SYSTEM LeGo2_0
  (* Version 1.0, Author, 4DIAC-Consortium *)
  APPLICATION HMI
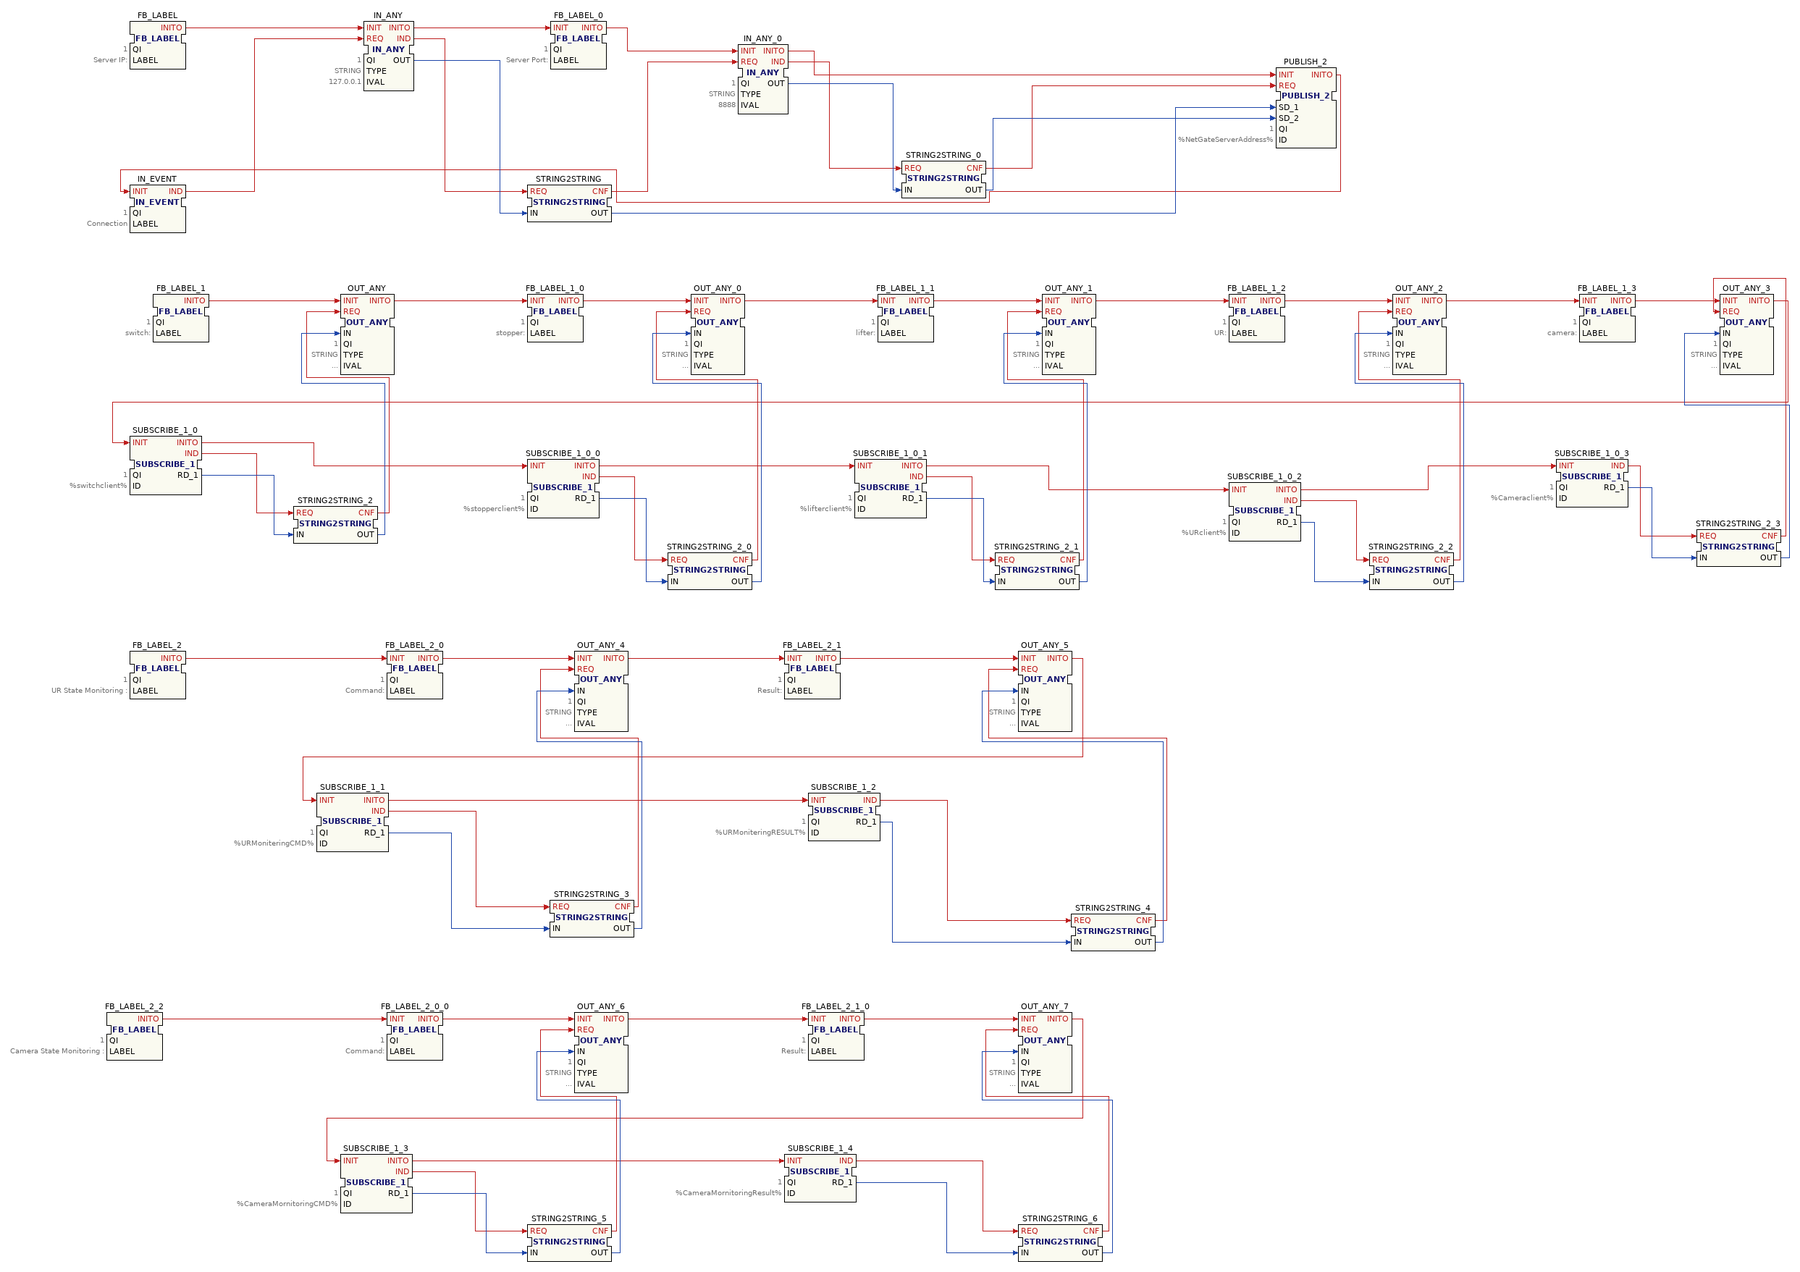
    FBS
      FB_LABEL : FB_LABEL(QI := 1, LABEL := Server IP:);
      FB_LABEL_0 : FB_LABEL(QI := 1, LABEL := Server Port:);
      IN_ANY : IN_ANY(QI := 1, TYPE := STRING, IVAL := 127.0.0.1);
      IN_ANY_0 : IN_ANY(QI := 1, TYPE := STRING, IVAL := 8888);
      PUBLISH_2 : PUBLISH_2(QI := 1, ID := %NetGateServerAddress%);
      STRING2STRING : STRING2STRING;
      STRING2STRING_0 : STRING2STRING;
      IN_EVENT : IN_EVENT(QI := 1, LABEL := Connection);
      FB_LABEL_1 : FB_LABEL(QI := 1, LABEL := switch:);
      FB_LABEL_1_0 : FB_LABEL(QI := 1, LABEL := stopper:);
      FB_LABEL_1_1 : FB_LABEL(QI := 1, LABEL := lifter:);
      FB_LABEL_1_2 : FB_LABEL(QI := 1, LABEL := UR:);
      FB_LABEL_1_3 : FB_LABEL(QI := 1, LABEL := camera:);
      OUT_ANY : OUT_ANY(QI := 1, TYPE := STRING, IVAL := ...);
      OUT_ANY_0 : OUT_ANY(QI := 1, TYPE := STRING, IVAL := ...);
      OUT_ANY_1 : OUT_ANY(QI := 1, TYPE := STRING, IVAL := ...);
      OUT_ANY_2 : OUT_ANY(QI := 1, TYPE := STRING, IVAL := ...);
      OUT_ANY_3 : OUT_ANY(QI := 1, TYPE := STRING, IVAL := ...);
      SUBSCRIBE_1_0 : SUBSCRIBE_1(QI := 1, ID := %switchclient%);
      SUBSCRIBE_1_0_0 : SUBSCRIBE_1(QI := 1, ID := %stopperclient%);
      SUBSCRIBE_1_0_1 : SUBSCRIBE_1(QI := 1, ID := %lifterclient%);
      SUBSCRIBE_1_0_2 : SUBSCRIBE_1(QI := 1, ID := %URclient%);
      SUBSCRIBE_1_0_3 : SUBSCRIBE_1(QI := 1, ID := %Cameraclient%);
      STRING2STRING_2 : STRING2STRING;
      STRING2STRING_2_0 : STRING2STRING;
      STRING2STRING_2_1 : STRING2STRING;
      STRING2STRING_2_2 : STRING2STRING;
      STRING2STRING_2_3 : STRING2STRING;
      FB_LABEL_2 : FB_LABEL(QI := 1, LABEL := UR State Monitoring :);
      FB_LABEL_2_0 : FB_LABEL(QI := 1, LABEL := Command:);
      FB_LABEL_2_1 : FB_LABEL(QI := 1, LABEL := Result:);
      FB_LABEL_2_2 : FB_LABEL(QI := 1, LABEL := Camera State Monitoring :);
      FB_LABEL_2_0_0 : FB_LABEL(QI := 1, LABEL := Command:);
      FB_LABEL_2_1_0 : FB_LABEL(QI := 1, LABEL := Result:);
      OUT_ANY_4 : OUT_ANY(QI := 1, TYPE := STRING, IVAL := ...);
      OUT_ANY_5 : OUT_ANY(QI := 1, TYPE := STRING, IVAL := ...);
      OUT_ANY_6 : OUT_ANY(QI := 1, TYPE := STRING, IVAL := ...);
      OUT_ANY_7 : OUT_ANY(QI := 1, TYPE := STRING, IVAL := ...);
      SUBSCRIBE_1_1 : SUBSCRIBE_1(QI := 1, ID := %URMoniteringCMD%);
      SUBSCRIBE_1_2 : SUBSCRIBE_1(QI := 1, ID := %URMoniteringRESULT%);
      SUBSCRIBE_1_3 : SUBSCRIBE_1(QI := 1, ID := %CameraMornitoringCMD%);
      SUBSCRIBE_1_4 : SUBSCRIBE_1(QI := 1, ID := %CameraMornitoringResult%);
      STRING2STRING_3 : STRING2STRING;
      STRING2STRING_4 : STRING2STRING;
      STRING2STRING_5 : STRING2STRING;
      STRING2STRING_6 : STRING2STRING;
    END_FBS
    EVENT_CONNECTIONS
      FB_LABEL.INITO TO IN_ANY.INIT;
      IN_ANY.INITO TO FB_LABEL_0.INIT;
      FB_LABEL_0.INITO TO IN_ANY_0.INIT;
      IN_ANY_0.INITO TO PUBLISH_2.INIT;
      IN_ANY.IND TO STRING2STRING.REQ;
      STRING2STRING.CNF TO IN_ANY_0.REQ;
      IN_ANY_0.IND TO STRING2STRING_0.REQ;
      STRING2STRING_0.CNF TO PUBLISH_2.REQ;
      IN_EVENT.IND TO IN_ANY.REQ;
      PUBLISH_2.INITO TO IN_EVENT.INIT;
      FB_LABEL_1.INITO TO OUT_ANY.INIT;
      OUT_ANY.INITO TO FB_LABEL_1_0.INIT;
      FB_LABEL_1_0.INITO TO OUT_ANY_0.INIT;
      OUT_ANY_0.INITO TO FB_LABEL_1_1.INIT;
      FB_LABEL_1_1.INITO TO OUT_ANY_1.INIT;
      OUT_ANY_1.INITO TO FB_LABEL_1_2.INIT;
      FB_LABEL_1_2.INITO TO OUT_ANY_2.INIT;
      OUT_ANY_2.INITO TO FB_LABEL_1_3.INIT;
      FB_LABEL_1_3.INITO TO OUT_ANY_3.INIT;
      OUT_ANY_3.INITO TO SUBSCRIBE_1_0.INIT;
      SUBSCRIBE_1_0.INITO TO SUBSCRIBE_1_0_0.INIT;
      SUBSCRIBE_1_0_0.INITO TO SUBSCRIBE_1_0_1.INIT;
      SUBSCRIBE_1_0_1.INITO TO SUBSCRIBE_1_0_2.INIT;
      SUBSCRIBE_1_0_2.INITO TO SUBSCRIBE_1_0_3.INIT;
      SUBSCRIBE_1_0.IND TO STRING2STRING_2.REQ;
      STRING2STRING_2.CNF TO OUT_ANY.REQ;
      SUBSCRIBE_1_0_0.IND TO STRING2STRING_2_0.REQ;
      STRING2STRING_2_0.CNF TO OUT_ANY_0.REQ;
      SUBSCRIBE_1_0_1.IND TO STRING2STRING_2_1.REQ;
      STRING2STRING_2_1.CNF TO OUT_ANY_1.REQ;
      SUBSCRIBE_1_0_2.IND TO STRING2STRING_2_2.REQ;
      STRING2STRING_2_2.CNF TO OUT_ANY_2.REQ;
      SUBSCRIBE_1_0_3.IND TO STRING2STRING_2_3.REQ;
      STRING2STRING_2_3.CNF TO OUT_ANY_3.REQ;
      FB_LABEL_2.INITO TO FB_LABEL_2_0.INIT;
      FB_LABEL_2_0.INITO TO OUT_ANY_4.INIT;
      OUT_ANY_4.INITO TO FB_LABEL_2_1.INIT;
      FB_LABEL_2_1.INITO TO OUT_ANY_5.INIT;
      FB_LABEL_2_2.INITO TO FB_LABEL_2_0_0.INIT;
      FB_LABEL_2_0_0.INITO TO OUT_ANY_6.INIT;
      OUT_ANY_6.INITO TO FB_LABEL_2_1_0.INIT;
      FB_LABEL_2_1_0.INITO TO OUT_ANY_7.INIT;
      OUT_ANY_5.INITO TO SUBSCRIBE_1_1.INIT;
      SUBSCRIBE_1_1.INITO TO SUBSCRIBE_1_2.INIT;
      SUBSCRIBE_1_1.IND TO STRING2STRING_3.REQ;
      STRING2STRING_3.CNF TO OUT_ANY_4.REQ;
      SUBSCRIBE_1_2.IND TO STRING2STRING_4.REQ;
      STRING2STRING_4.CNF TO OUT_ANY_5.REQ;
      OUT_ANY_7.INITO TO SUBSCRIBE_1_3.INIT;
      SUBSCRIBE_1_3.INITO TO SUBSCRIBE_1_4.INIT;
      SUBSCRIBE_1_3.IND TO STRING2STRING_5.REQ;
      STRING2STRING_5.CNF TO OUT_ANY_6.REQ;
      SUBSCRIBE_1_4.IND TO STRING2STRING_6.REQ;
      STRING2STRING_6.CNF TO OUT_ANY_7.REQ;
    END_CONNECTIONS
    DATA_CONNECTIONS
      IN_ANY.OUT TO STRING2STRING.IN;
      STRING2STRING.OUT TO PUBLISH_2.SD_1;
      IN_ANY_0.OUT TO STRING2STRING_0.IN;
      STRING2STRING_0.OUT TO PUBLISH_2.SD_2;
      SUBSCRIBE_1_0.RD_1 TO STRING2STRING_2.IN;
      STRING2STRING_2.OUT TO OUT_ANY.IN;
      SUBSCRIBE_1_0_0.RD_1 TO STRING2STRING_2_0.IN;
      STRING2STRING_2_0.OUT TO OUT_ANY_0.IN;
      SUBSCRIBE_1_0_1.RD_1 TO STRING2STRING_2_1.IN;
      STRING2STRING_2_1.OUT TO OUT_ANY_1.IN;
      SUBSCRIBE_1_0_2.RD_1 TO STRING2STRING_2_2.IN;
      STRING2STRING_2_2.OUT TO OUT_ANY_2.IN;
      SUBSCRIBE_1_0_3.RD_1 TO STRING2STRING_2_3.IN;
      STRING2STRING_2_3.OUT TO OUT_ANY_3.IN;
      SUBSCRIBE_1_1.RD_1 TO STRING2STRING_3.IN;
      STRING2STRING_3.OUT TO OUT_ANY_4.IN;
      SUBSCRIBE_1_2.RD_1 TO STRING2STRING_4.IN;
      STRING2STRING_4.OUT TO OUT_ANY_5.IN;
      SUBSCRIBE_1_3.RD_1 TO STRING2STRING_5.IN;
      STRING2STRING_5.OUT TO OUT_ANY_6.IN;
      SUBSCRIBE_1_4.RD_1 TO STRING2STRING_6.IN;
      STRING2STRING_6.OUT TO OUT_ANY_7.IN;
    END_CONNECTIONS
  END_APPLICATION
  APPLICATION SwitchStopperLifter
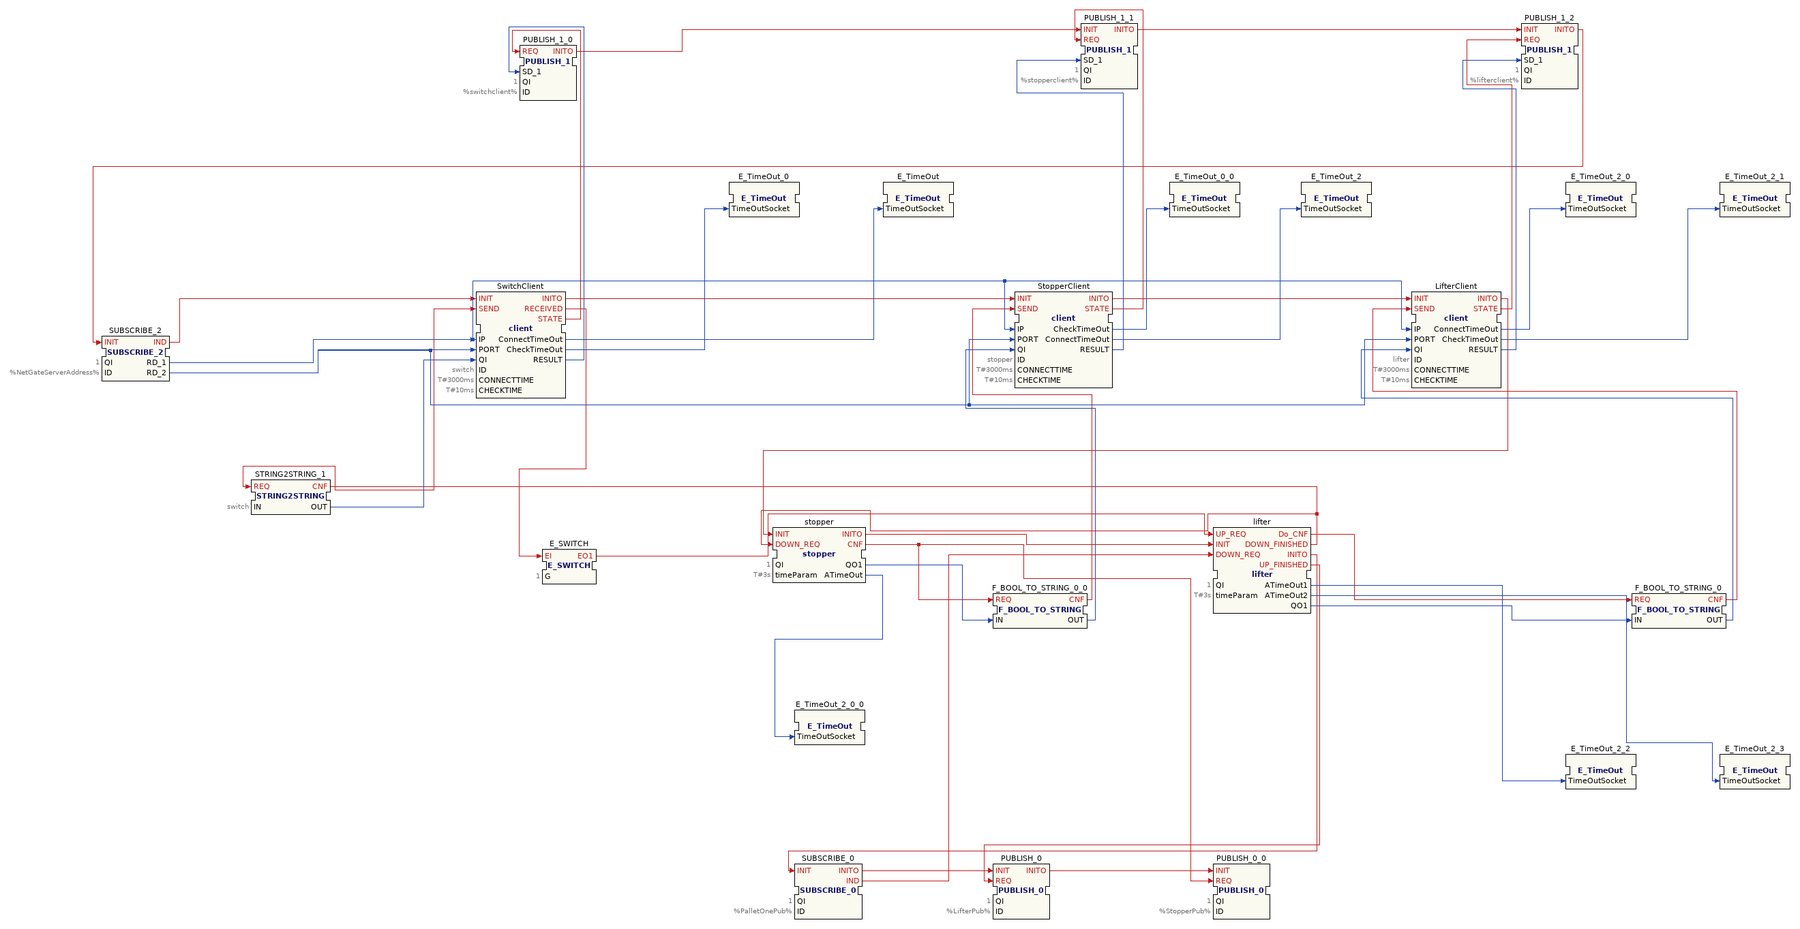
    FBS
      SwitchClient : client(ID := switch, CONNECTTIME := T#3000ms, CHECKTIME := T#10ms);
      E_TimeOut : E_TimeOut;
      E_TimeOut_0 : E_TimeOut;
      SUBSCRIBE_2 : SUBSCRIBE_2(QI := 1, ID := %NetGateServerAddress%);
      LifterClient : client(ID := lifter, CONNECTTIME := T#3000ms, CHECKTIME := T#10ms);
      E_TimeOut_0_0 : E_TimeOut;
      StopperClient : client(ID := stopper, CONNECTTIME := T#3000ms, CHECKTIME := T#10ms);
      E_TimeOut_2 : E_TimeOut;
      E_SWITCH : E_SWITCH(G := 1);
      stopper : stopper(QI := 1, timeParam := T#3s);
      lifter : lifter(QI := 1, timeParam := T#3s);
      E_TimeOut_2_0 : E_TimeOut;
      E_TimeOut_2_1 : E_TimeOut;
      E_TimeOut_2_2 : E_TimeOut;
      E_TimeOut_2_3 : E_TimeOut;
      F_BOOL_TO_STRING_0 : F_BOOL_TO_STRING;
      F_BOOL_TO_STRING_0_0 : F_BOOL_TO_STRING;
      E_TimeOut_2_0_0 : E_TimeOut;
      STRING2STRING_1 : STRING2STRING(IN := switch);
      PUBLISH_0 : PUBLISH_0(QI := 1, ID := %LifterPub%);
      SUBSCRIBE_0 : SUBSCRIBE_0(QI := 1, ID := %PalletOnePub%);
      PUBLISH_0_0 : PUBLISH_0(QI := 1, ID := %StopperPub%);
      PUBLISH_1_0 : PUBLISH_1(QI := 1, ID := %switchclient%);
      PUBLISH_1_1 : PUBLISH_1(QI := 1, ID := %stopperclient%);
      PUBLISH_1_2 : PUBLISH_1(QI := 1, ID := %lifterclient%);
    END_FBS
    EVENT_CONNECTIONS
      SUBSCRIBE_2.IND TO SwitchClient.INIT;
      SwitchClient.INITO TO StopperClient.INIT;
      StopperClient.INITO TO LifterClient.INIT;
      SwitchClient.RECEIVED TO E_SWITCH.EI;
      E_SWITCH.EO1 TO lifter.UP_REQ;
      LifterClient.INITO TO stopper.INIT;
      stopper.INITO TO lifter.INIT;
      lifter.Do_CNF TO F_BOOL_TO_STRING_0.REQ;
      F_BOOL_TO_STRING_0.CNF TO LifterClient.SEND;
      stopper.CNF TO F_BOOL_TO_STRING_0_0.REQ;
      F_BOOL_TO_STRING_0_0.CNF TO StopperClient.SEND;
      lifter.DOWN_FINISHED TO stopper.DOWN_REQ;
      lifter.DOWN_FINISHED TO STRING2STRING_1.REQ;
      STRING2STRING_1.CNF TO SwitchClient.SEND;
      lifter.INITO TO SUBSCRIBE_0.INIT;
      SUBSCRIBE_0.INITO TO PUBLISH_0.INIT;
      SUBSCRIBE_0.IND TO lifter.DOWN_REQ;
      lifter.UP_FINISHED TO PUBLISH_0.REQ;
      PUBLISH_0.INITO TO PUBLISH_0_0.INIT;
      stopper.CNF TO PUBLISH_0_0.REQ;
      PUBLISH_1_0.INITO TO PUBLISH_1_1.INIT;
      PUBLISH_1_1.INITO TO PUBLISH_1_2.INIT;
      PUBLISH_1_2.INITO TO SUBSCRIBE_2.INIT;
      SwitchClient.STATE TO PUBLISH_1_0.REQ;
      StopperClient.STATE TO PUBLISH_1_1.REQ;
      LifterClient.STATE TO PUBLISH_1_2.REQ;
    END_CONNECTIONS
    DATA_CONNECTIONS
      SwitchClient.ConnectTimeOut TO E_TimeOut.TimeOutSocket;
      SwitchClient.CheckTimeOut TO E_TimeOut_0.TimeOutSocket;
      SUBSCRIBE_2.RD_1 TO SwitchClient.IP;
      SUBSCRIBE_2.RD_2 TO SwitchClient.PORT;
      SUBSCRIBE_2.RD_1 TO LifterClient.IP;
      SUBSCRIBE_2.RD_2 TO LifterClient.PORT;
      StopperClient.CheckTimeOut TO E_TimeOut_0_0.TimeOutSocket;
      StopperClient.ConnectTimeOut TO E_TimeOut_2.TimeOutSocket;
      SUBSCRIBE_2.RD_1 TO StopperClient.IP;
      SUBSCRIBE_2.RD_2 TO StopperClient.PORT;
      LifterClient.ConnectTimeOut TO E_TimeOut_2_0.TimeOutSocket;
      LifterClient.CheckTimeOut TO E_TimeOut_2_1.TimeOutSocket;
      lifter.ATimeOut1 TO E_TimeOut_2_2.TimeOutSocket;
      lifter.ATimeOut2 TO E_TimeOut_2_3.TimeOutSocket;
      lifter.QO1 TO F_BOOL_TO_STRING_0.IN;
      F_BOOL_TO_STRING_0.OUT TO LifterClient.QI;
      stopper.QO1 TO F_BOOL_TO_STRING_0_0.IN;
      F_BOOL_TO_STRING_0_0.OUT TO StopperClient.QI;
      stopper.ATimeOut TO E_TimeOut_2_0_0.TimeOutSocket;
      STRING2STRING_1.OUT TO SwitchClient.QI;
      SwitchClient.RESULT TO PUBLISH_1_0.SD_1;
      StopperClient.RESULT TO PUBLISH_1_1.SD_1;
      LifterClient.RESULT TO PUBLISH_1_2.SD_1;
    END_CONNECTIONS
  END_APPLICATION
  APPLICATION URCamera
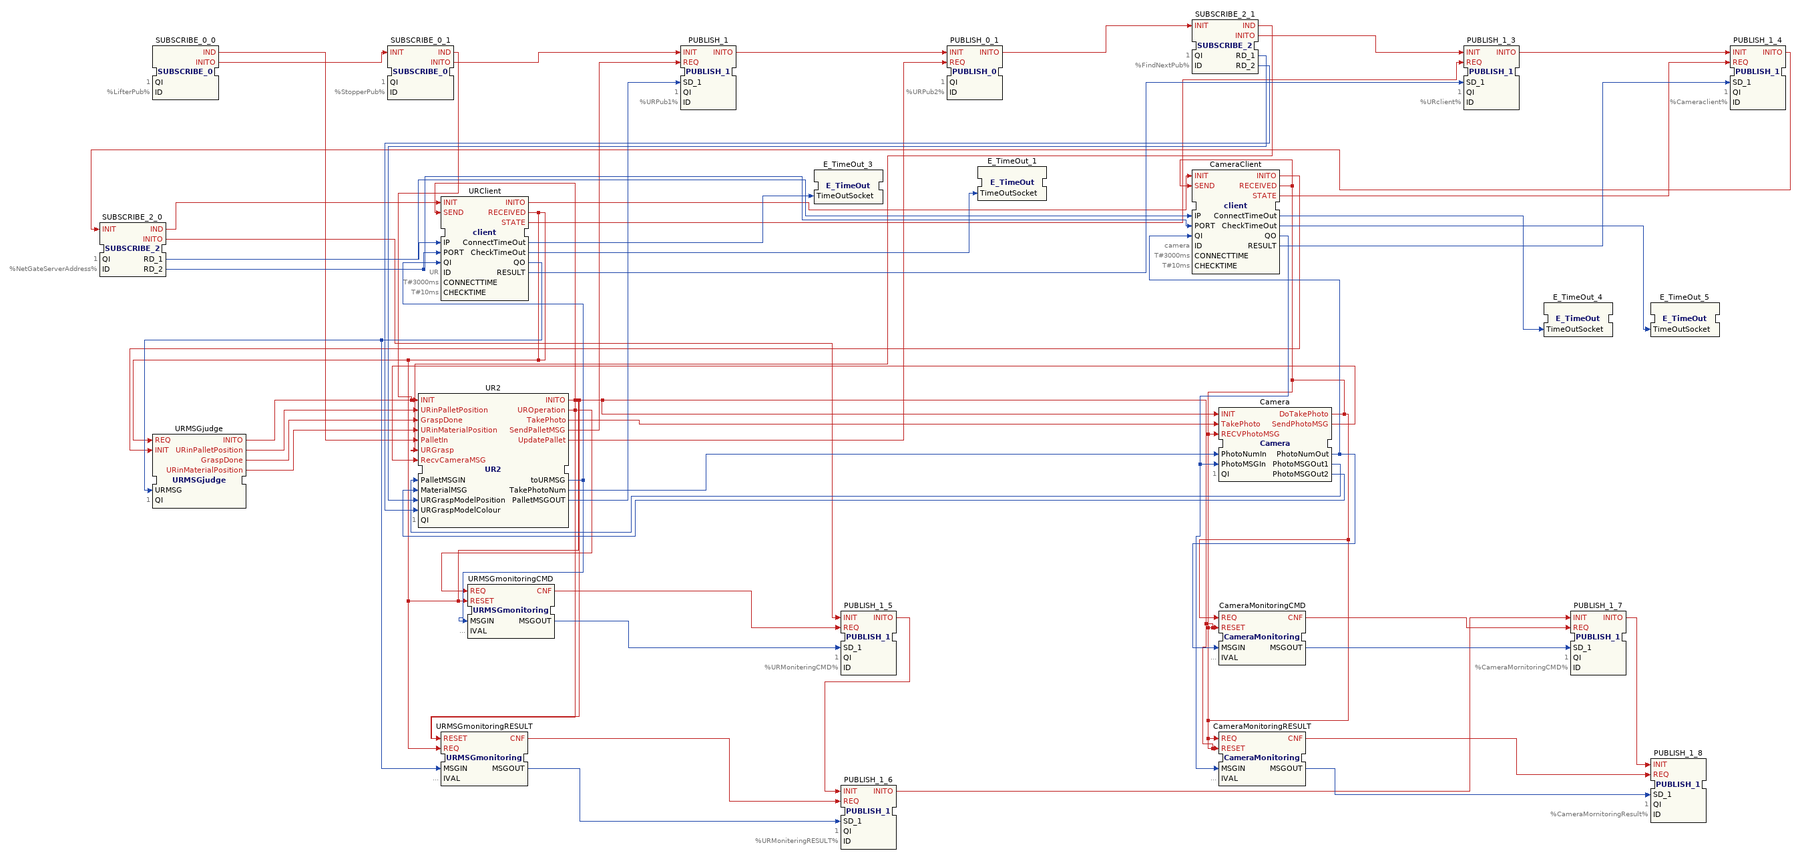
    FBS
      UR2 : UR2(QI := 1);
      URMSGjudge : URMSGjudge(QI := 1);
      URMSGmonitoringRESULT : URMSGmonitoring(IVAL := ...);
      URClient : client(ID := UR, CONNECTTIME := T#3000ms, CHECKTIME := T#10ms);
      E_TimeOut_1 : E_TimeOut;
      E_TimeOut_3 : E_TimeOut;
      Camera : Camera(QI := 1);
      CameraMonitoringCMD : CameraMonitoring(IVAL := ...);
      CameraClient : client(ID := camera, CONNECTTIME := T#3000ms, CHECKTIME := T#10ms);
      E_TimeOut_4 : E_TimeOut;
      E_TimeOut_5 : E_TimeOut;
      SUBSCRIBE_2_0 : SUBSCRIBE_2(QI := 1, ID := %NetGateServerAddress%);
      SUBSCRIBE_0_0 : SUBSCRIBE_0(QI := 1, ID := %LifterPub%);
      SUBSCRIBE_0_1 : SUBSCRIBE_0(QI := 1, ID := %StopperPub%);
      PUBLISH_1 : PUBLISH_1(QI := 1, ID := %URPub1%);
      PUBLISH_0_1 : PUBLISH_0(QI := 1, ID := %URPub2%);
      SUBSCRIBE_2_1 : SUBSCRIBE_2(QI := 1, ID := %FindNextPub%);
      PUBLISH_1_3 : PUBLISH_1(QI := 1, ID := %URclient%);
      PUBLISH_1_4 : PUBLISH_1(QI := 1, ID := %Cameraclient%);
      URMSGmonitoringCMD : URMSGmonitoring(IVAL := ...);
      CameraMonitoringRESULT : CameraMonitoring(IVAL := ...);
      PUBLISH_1_5 : PUBLISH_1(QI := 1, ID := %URMoniteringCMD%);
      PUBLISH_1_6 : PUBLISH_1(QI := 1, ID := %URMoniteringRESULT%);
      PUBLISH_1_7 : PUBLISH_1(QI := 1, ID := %CameraMornitoringCMD%);
      PUBLISH_1_8 : PUBLISH_1(QI := 1, ID := %CameraMornitoringResult%);
    END_FBS
    EVENT_CONNECTIONS
      SUBSCRIBE_2_0.IND TO URClient.INIT;
      URClient.INITO TO CameraClient.INIT;
      URClient.RECEIVED TO URMSGjudge.REQ;
      CameraClient.INITO TO URMSGjudge.INIT;
      URMSGjudge.INITO TO UR2.INIT;
      UR2.INITO TO Camera.INIT;
      URMSGjudge.URinPalletPosition TO UR2.URinPalletPosition;
      URMSGjudge.GraspDone TO UR2.GraspDone;
      URMSGjudge.URinMaterialPosition TO UR2.URinMaterialPosition;
      SUBSCRIBE_0_0.IND TO UR2.PalletIn;
      SUBSCRIBE_0_0.INITO TO SUBSCRIBE_0_1.INIT;
      SUBSCRIBE_0_1.IND TO UR2.INIT;
      UR2.UROperation TO URClient.SEND;
      UR2.TakePhoto TO Camera.TakePhoto;
      Camera.DoTakePhoto TO CameraClient.SEND;
      CameraClient.RECEIVED TO Camera.RECVPhotoMSG;
      SUBSCRIBE_0_1.INITO TO PUBLISH_1.INIT;
      PUBLISH_1.INITO TO PUBLISH_0_1.INIT;
      UR2.SendPalletMSG TO PUBLISH_1.REQ;
      UR2.UpdatePallet TO PUBLISH_0_1.REQ;
      PUBLISH_0_1.INITO TO SUBSCRIBE_2_1.INIT;
      SUBSCRIBE_2_1.IND TO UR2.URGrasp;
      Camera.SendPhotoMSG TO UR2.RecvCameraMSG;
      SUBSCRIBE_2_1.INITO TO PUBLISH_1_3.INIT;
      PUBLISH_1_3.INITO TO PUBLISH_1_4.INIT;
      URClient.STATE TO PUBLISH_1_3.REQ;
      CameraClient.STATE TO PUBLISH_1_4.REQ;
      PUBLISH_1_4.INITO TO SUBSCRIBE_2_0.INIT;
      UR2.UROperation TO URMSGmonitoringCMD.REQ;
      UR2.UROperation TO URMSGmonitoringRESULT.RESET;
      URClient.RECEIVED TO URMSGmonitoringRESULT.REQ;
      URClient.RECEIVED TO URMSGmonitoringCMD.RESET;
      Camera.DoTakePhoto TO CameraMonitoringCMD.REQ;
      CameraClient.RECEIVED TO CameraMonitoringRESULT.REQ;
      Camera.DoTakePhoto TO CameraMonitoringRESULT.RESET;
      CameraClient.RECEIVED TO CameraMonitoringCMD.RESET;
      SUBSCRIBE_2_0.INITO TO PUBLISH_1_5.INIT;
      PUBLISH_1_5.INITO TO PUBLISH_1_6.INIT;
      PUBLISH_1_6.INITO TO PUBLISH_1_7.INIT;
      PUBLISH_1_7.INITO TO PUBLISH_1_8.INIT;
      URMSGmonitoringCMD.CNF TO PUBLISH_1_5.REQ;
      URMSGmonitoringRESULT.CNF TO PUBLISH_1_6.REQ;
      CameraMonitoringCMD.CNF TO PUBLISH_1_7.REQ;
      CameraMonitoringRESULT.CNF TO PUBLISH_1_8.REQ;
      UR2.INITO TO URMSGmonitoringCMD.RESET;
      UR2.INITO TO URMSGmonitoringRESULT.RESET;
      UR2.INITO TO CameraMonitoringCMD.RESET;
      UR2.INITO TO CameraMonitoringRESULT.RESET;
    END_CONNECTIONS
    DATA_CONNECTIONS
      URClient.ConnectTimeOut TO E_TimeOut_3.TimeOutSocket;
      URClient.CheckTimeOut TO E_TimeOut_1.TimeOutSocket;
      CameraClient.ConnectTimeOut TO E_TimeOut_4.TimeOutSocket;
      CameraClient.CheckTimeOut TO E_TimeOut_5.TimeOutSocket;
      SUBSCRIBE_2_0.RD_1 TO URClient.IP;
      SUBSCRIBE_2_0.RD_2 TO URClient.PORT;
      SUBSCRIBE_2_0.RD_1 TO CameraClient.IP;
      SUBSCRIBE_2_0.RD_2 TO CameraClient.PORT;
      URClient.QO TO URMSGjudge.URMSG;
      UR2.toURMSG TO URClient.QI;
      UR2.TakePhotoNum TO Camera.PhotoNumIn;
      Camera.PhotoNumOut TO CameraClient.QI;
      CameraClient.QO TO Camera.PhotoMSGIn;
      Camera.PhotoMSGOut1 TO UR2.PalletMSGIN;
      Camera.PhotoMSGOut2 TO UR2.MaterialMSG;
      UR2.PalletMSGOUT TO PUBLISH_1.SD_1;
      SUBSCRIBE_2_1.RD_1 TO UR2.URGraspModelPosition;
      SUBSCRIBE_2_1.RD_2 TO UR2.URGraspModelColour;
      URClient.RESULT TO PUBLISH_1_3.SD_1;
      CameraClient.RESULT TO PUBLISH_1_4.SD_1;
      UR2.toURMSG TO URMSGmonitoringCMD.MSGIN;
      URClient.QO TO URMSGmonitoringRESULT.MSGIN;
      Camera.PhotoNumOut TO CameraMonitoringCMD.MSGIN;
      CameraClient.QO TO CameraMonitoringRESULT.MSGIN;
      URMSGmonitoringCMD.MSGOUT TO PUBLISH_1_5.SD_1;
      URMSGmonitoringRESULT.MSGOUT TO PUBLISH_1_6.SD_1;
      CameraMonitoringCMD.MSGOUT TO PUBLISH_1_7.SD_1;
      CameraMonitoringRESULT.MSGOUT TO PUBLISH_1_8.SD_1;
    END_CONNECTIONS
  END_APPLICATION
  APPLICATION DataBaseOperation
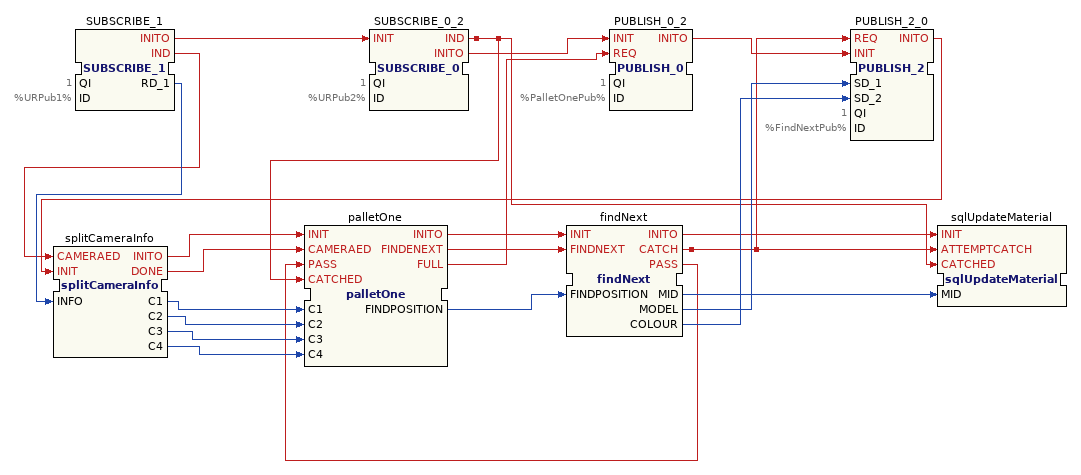
    FBS
      sqlUpdateMaterial : sqlUpdateMaterial;
      splitCameraInfo : splitCameraInfo;
      findNext : findNext;
      palletOne : palletOne;
      SUBSCRIBE_0_2 : SUBSCRIBE_0(QI := 1, ID := %URPub2%);
      SUBSCRIBE_1 : SUBSCRIBE_1(QI := 1, ID := %URPub1%);
      PUBLISH_2_0 : PUBLISH_2(QI := 1, ID := %FindNextPub%);
      PUBLISH_0_2 : PUBLISH_0(QI := 1, ID := %PalletOnePub%);
    END_FBS
    EVENT_CONNECTIONS
      findNext.INITO TO sqlUpdateMaterial.INIT;
      splitCameraInfo.INITO TO palletOne.INIT;
      palletOne.INITO TO findNext.INIT;
      splitCameraInfo.DONE TO palletOne.CAMERAED;
      palletOne.FINDENEXT TO findNext.FINDNEXT;
      findNext.CATCH TO sqlUpdateMaterial.ATTEMPTCATCH;
      findNext.PASS TO palletOne.PASS;
      SUBSCRIBE_1.INITO TO SUBSCRIBE_0_2.INIT;
      SUBSCRIBE_1.IND TO splitCameraInfo.CAMERAED;
      SUBSCRIBE_0_2.IND TO palletOne.CATCHED;
      SUBSCRIBE_0_2.IND TO sqlUpdateMaterial.CATCHED;
      findNext.CATCH TO PUBLISH_2_0.REQ;
      SUBSCRIBE_0_2.INITO TO PUBLISH_0_2.INIT;
      PUBLISH_0_2.INITO TO PUBLISH_2_0.INIT;
      PUBLISH_2_0.INITO TO splitCameraInfo.INIT;
      palletOne.FULL TO PUBLISH_0_2.REQ;
    END_CONNECTIONS
    DATA_CONNECTIONS
      splitCameraInfo.C1 TO palletOne.C1;
      splitCameraInfo.C2 TO palletOne.C2;
      splitCameraInfo.C3 TO palletOne.C3;
      splitCameraInfo.C4 TO palletOne.C4;
      findNext.MID TO sqlUpdateMaterial.MID;
      findNext.MODEL TO PUBLISH_2_0.SD_1;
      findNext.COLOUR TO PUBLISH_2_0.SD_2;
      SUBSCRIBE_1.RD_1 TO splitCameraInfo.INFO;
      palletOne.FINDPOSITION TO findNext.FINDPOSITION;
    END_CONNECTIONS
  END_APPLICATION
  DEVICE FORTE_PC : FORTE_PC(MGR_ID := "192.168.1.100:61499")
    {SET_ATTRIBUTE(Profile, HOLOBLOC)}
    RESOURCE EMB_RES : EMB_RES
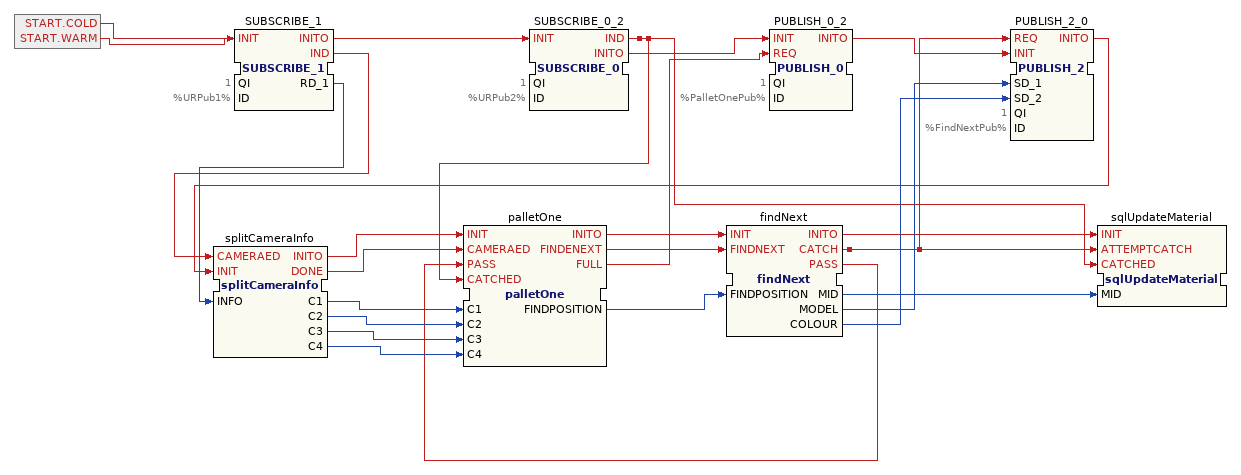
      FBS
        sqlUpdateMaterial : sqlUpdateMaterial;
        splitCameraInfo : splitCameraInfo;
        findNext : findNext;
        palletOne : palletOne;
        SUBSCRIBE_0_2 : SUBSCRIBE_0(QI := 1, ID := %URPub2%);
        SUBSCRIBE_1 : SUBSCRIBE_1(QI := 1, ID := %URPub1%);
        PUBLISH_2_0 : PUBLISH_2(QI := 1, ID := %FindNextPub%);
        PUBLISH_0_2 : PUBLISH_0(QI := 1, ID := %PalletOnePub%);
      END_FBS
      EVENT_CONNECTIONS
        findNext.INITO TO sqlUpdateMaterial.INIT;
        findNext.CATCH TO sqlUpdateMaterial.ATTEMPTCATCH;
        splitCameraInfo.INITO TO palletOne.INIT;
        splitCameraInfo.DONE TO palletOne.CAMERAED;
        findNext.PASS TO palletOne.PASS;
        palletOne.INITO TO findNext.INIT;
        palletOne.FINDENEXT TO findNext.FINDNEXT;
        SUBSCRIBE_0_2.IND TO palletOne.CATCHED;
        SUBSCRIBE_0_2.IND TO sqlUpdateMaterial.CATCHED;
        SUBSCRIBE_1.INITO TO SUBSCRIBE_0_2.INIT;
        SUBSCRIBE_1.IND TO splitCameraInfo.CAMERAED;
        findNext.CATCH TO PUBLISH_2_0.REQ;
        PUBLISH_2_0.INITO TO splitCameraInfo.INIT;
        SUBSCRIBE_0_2.INITO TO PUBLISH_0_2.INIT;
        palletOne.FULL TO PUBLISH_0_2.REQ;
        PUBLISH_0_2.INITO TO PUBLISH_2_0.INIT;
        START.COLD TO SUBSCRIBE_1.INIT;
        START.WARM TO SUBSCRIBE_1.INIT;
      END_CONNECTIONS
      DATA_CONNECTIONS
        findNext.MID TO sqlUpdateMaterial.MID;
        splitCameraInfo.C1 TO palletOne.C1;
        splitCameraInfo.C2 TO palletOne.C2;
        splitCameraInfo.C3 TO palletOne.C3;
        splitCameraInfo.C4 TO palletOne.C4;
        SUBSCRIBE_1.RD_1 TO splitCameraInfo.INFO;
        findNext.MODEL TO PUBLISH_2_0.SD_1;
        findNext.COLOUR TO PUBLISH_2_0.SD_2;
        palletOne.FINDPOSITION TO findNext.FINDPOSITION;
      END_CONNECTIONS
    END_RESOURCE
  END_DEVICE
  DEVICE FBRT_WINDOW : FBRT_WINDOW(MGR_ID := "192.168.1.100:61505")
    {SET_ATTRIBUTE(Profile, HOLOBLOC)}
    RESOURCE ConnectSet : PANEL_RESOURCE
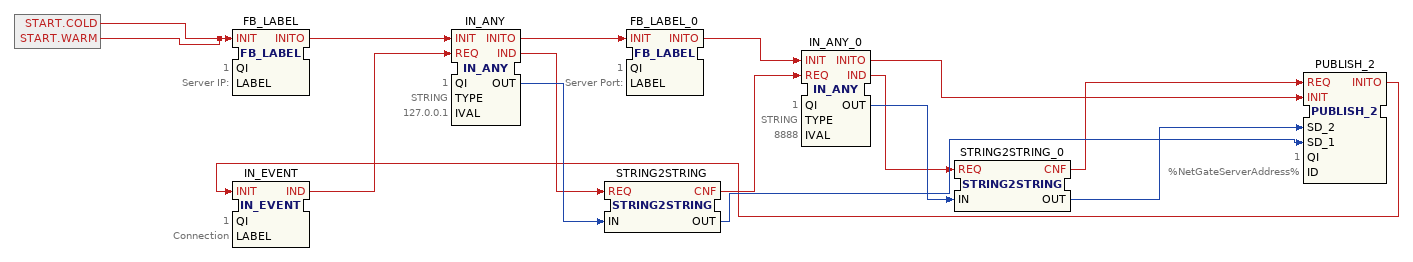
      FBS
        FB_LABEL : FB_LABEL(QI := 1, LABEL := Server IP:);
        PUBLISH_2 : PUBLISH_2(QI := 1, ID := %NetGateServerAddress%);
        FB_LABEL_0 : FB_LABEL(QI := 1, LABEL := Server Port:);
        STRING2STRING_0 : STRING2STRING;
        IN_ANY : IN_ANY(QI := 1, TYPE := STRING, IVAL := 127.0.0.1);
        STRING2STRING : STRING2STRING;
        IN_EVENT : IN_EVENT(QI := 1, LABEL := Connection);
        IN_ANY_0 : IN_ANY(QI := 1, TYPE := STRING, IVAL := 8888);
      END_FBS
      EVENT_CONNECTIONS
        STRING2STRING_0.CNF TO PUBLISH_2.REQ;
        FB_LABEL.INITO TO IN_ANY.INIT;
        IN_ANY.INITO TO FB_LABEL_0.INIT;
        IN_ANY.IND TO STRING2STRING.REQ;
        PUBLISH_2.INITO TO IN_EVENT.INIT;
        IN_EVENT.IND TO IN_ANY.REQ;
        FB_LABEL_0.INITO TO IN_ANY_0.INIT;
        STRING2STRING.CNF TO IN_ANY_0.REQ;
        IN_ANY_0.INITO TO PUBLISH_2.INIT;
        IN_ANY_0.IND TO STRING2STRING_0.REQ;
        START.COLD TO FB_LABEL.INIT;
        START.WARM TO FB_LABEL.INIT;
      END_CONNECTIONS
      DATA_CONNECTIONS
        STRING2STRING_0.OUT TO PUBLISH_2.SD_2;
        IN_ANY.OUT TO STRING2STRING.IN;
        STRING2STRING.OUT TO PUBLISH_2.SD_1;
        IN_ANY_0.OUT TO STRING2STRING_0.IN;
      END_CONNECTIONS
    END_RESOURCE
    RESOURCE ClientConnection : PANEL_RESOURCE
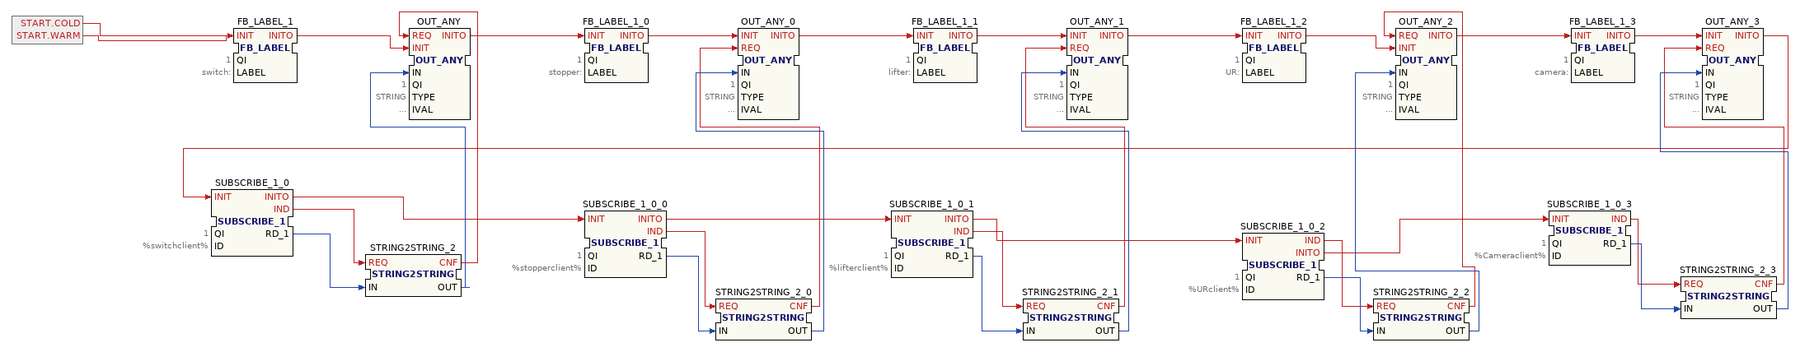
      FBS
        OUT_ANY_2 : OUT_ANY(QI := 1, TYPE := STRING, IVAL := ...);
        STRING2STRING_2_2 : STRING2STRING;
        STRING2STRING_2_1 : STRING2STRING;
        STRING2STRING_2_0 : STRING2STRING;
        FB_LABEL_1_0 : FB_LABEL(QI := 1, LABEL := stopper:);
        FB_LABEL_1_1 : FB_LABEL(QI := 1, LABEL := lifter:);
        SUBSCRIBE_1_0_2 : SUBSCRIBE_1(QI := 1, ID := %URclient%);
        SUBSCRIBE_1_0_1 : SUBSCRIBE_1(QI := 1, ID := %lifterclient%);
        OUT_ANY_0 : OUT_ANY(QI := 1, TYPE := STRING, IVAL := ...);
        STRING2STRING_2 : STRING2STRING;
        OUT_ANY_1 : OUT_ANY(QI := 1, TYPE := STRING, IVAL := ...);
        FB_LABEL_1_2 : FB_LABEL(QI := 1, LABEL := UR:);
        SUBSCRIBE_1_0_3 : SUBSCRIBE_1(QI := 1, ID := %Cameraclient%);
        OUT_ANY : OUT_ANY(QI := 1, TYPE := STRING, IVAL := ...);
        FB_LABEL_1 : FB_LABEL(QI := 1, LABEL := switch:);
        SUBSCRIBE_1_0_0 : SUBSCRIBE_1(QI := 1, ID := %stopperclient%);
        SUBSCRIBE_1_0 : SUBSCRIBE_1(QI := 1, ID := %switchclient%);
        FB_LABEL_1_3 : FB_LABEL(QI := 1, LABEL := camera:);
        OUT_ANY_3 : OUT_ANY(QI := 1, TYPE := STRING, IVAL := ...);
        STRING2STRING_2_3 : STRING2STRING;
      END_FBS
      EVENT_CONNECTIONS
        STRING2STRING_2_2.CNF TO OUT_ANY_2.REQ;
        SUBSCRIBE_1_0_2.IND TO STRING2STRING_2_2.REQ;
        SUBSCRIBE_1_0_1.INITO TO SUBSCRIBE_1_0_2.INIT;
        SUBSCRIBE_1_0_1.IND TO STRING2STRING_2_1.REQ;
        FB_LABEL_1_0.INITO TO OUT_ANY_0.INIT;
        STRING2STRING_2_0.CNF TO OUT_ANY_0.REQ;
        OUT_ANY_0.INITO TO FB_LABEL_1_1.INIT;
        FB_LABEL_1_1.INITO TO OUT_ANY_1.INIT;
        STRING2STRING_2_1.CNF TO OUT_ANY_1.REQ;
        OUT_ANY_1.INITO TO FB_LABEL_1_2.INIT;
        FB_LABEL_1_2.INITO TO OUT_ANY_2.INIT;
        SUBSCRIBE_1_0_2.INITO TO SUBSCRIBE_1_0_3.INIT;
        STRING2STRING_2.CNF TO OUT_ANY.REQ;
        OUT_ANY.INITO TO FB_LABEL_1_0.INIT;
        FB_LABEL_1.INITO TO OUT_ANY.INIT;
        SUBSCRIBE_1_0_0.INITO TO SUBSCRIBE_1_0_1.INIT;
        SUBSCRIBE_1_0_0.IND TO STRING2STRING_2_0.REQ;
        SUBSCRIBE_1_0.INITO TO SUBSCRIBE_1_0_0.INIT;
        SUBSCRIBE_1_0.IND TO STRING2STRING_2.REQ;
        OUT_ANY_2.INITO TO FB_LABEL_1_3.INIT;
        FB_LABEL_1_3.INITO TO OUT_ANY_3.INIT;
        OUT_ANY_3.INITO TO SUBSCRIBE_1_0.INIT;
        SUBSCRIBE_1_0_3.IND TO STRING2STRING_2_3.REQ;
        STRING2STRING_2_3.CNF TO OUT_ANY_3.REQ;
        START.COLD TO FB_LABEL_1.INIT;
        START.WARM TO FB_LABEL_1.INIT;
      END_CONNECTIONS
      DATA_CONNECTIONS
        STRING2STRING_2_2.OUT TO OUT_ANY_2.IN;
        SUBSCRIBE_1_0_2.RD_1 TO STRING2STRING_2_2.IN;
        SUBSCRIBE_1_0_1.RD_1 TO STRING2STRING_2_1.IN;
        STRING2STRING_2_0.OUT TO OUT_ANY_0.IN;
        STRING2STRING_2_1.OUT TO OUT_ANY_1.IN;
        STRING2STRING_2.OUT TO OUT_ANY.IN;
        SUBSCRIBE_1_0_0.RD_1 TO STRING2STRING_2_0.IN;
        SUBSCRIBE_1_0.RD_1 TO STRING2STRING_2.IN;
        SUBSCRIBE_1_0_3.RD_1 TO STRING2STRING_2_3.IN;
        STRING2STRING_2_3.OUT TO OUT_ANY_3.IN;
      END_CONNECTIONS
    END_RESOURCE
    RESOURCE MachineState : PANEL_RESOURCE
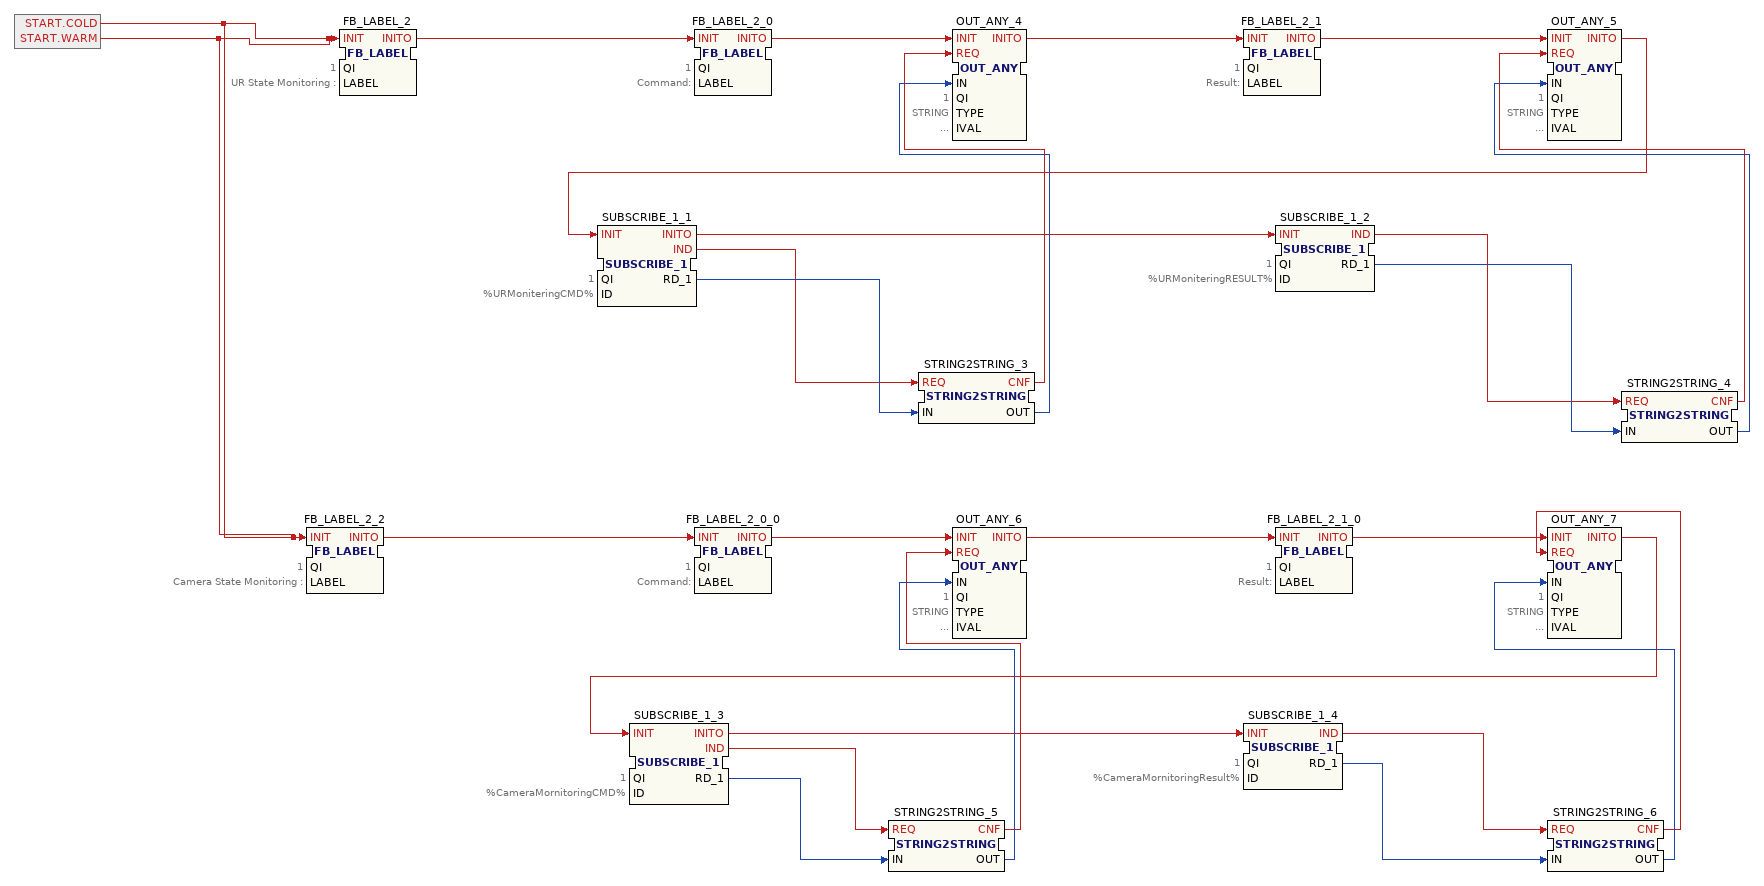
      FBS
        FB_LABEL_2 : FB_LABEL(QI := 1, LABEL := UR State Monitoring :);
        FB_LABEL_2_0 : FB_LABEL(QI := 1, LABEL := Command:);
        FB_LABEL_2_1 : FB_LABEL(QI := 1, LABEL := Result:);
        FB_LABEL_2_2 : FB_LABEL(QI := 1, LABEL := Camera State Monitoring :);
        FB_LABEL_2_0_0 : FB_LABEL(QI := 1, LABEL := Command:);
        FB_LABEL_2_1_0 : FB_LABEL(QI := 1, LABEL := Result:);
        OUT_ANY_4 : OUT_ANY(QI := 1, TYPE := STRING, IVAL := ...);
        OUT_ANY_5 : OUT_ANY(QI := 1, TYPE := STRING, IVAL := ...);
        OUT_ANY_6 : OUT_ANY(QI := 1, TYPE := STRING, IVAL := ...);
        OUT_ANY_7 : OUT_ANY(QI := 1, TYPE := STRING, IVAL := ...);
        SUBSCRIBE_1_1 : SUBSCRIBE_1(QI := 1, ID := %URMoniteringCMD%);
        SUBSCRIBE_1_2 : SUBSCRIBE_1(QI := 1, ID := %URMoniteringRESULT%);
        SUBSCRIBE_1_3 : SUBSCRIBE_1(QI := 1, ID := %CameraMornitoringCMD%);
        SUBSCRIBE_1_4 : SUBSCRIBE_1(QI := 1, ID := %CameraMornitoringResult%);
        STRING2STRING_3 : STRING2STRING;
        STRING2STRING_4 : STRING2STRING;
        STRING2STRING_5 : STRING2STRING;
        STRING2STRING_6 : STRING2STRING;
      END_FBS
      EVENT_CONNECTIONS
        FB_LABEL_2.INITO TO FB_LABEL_2_0.INIT;
        FB_LABEL_2_2.INITO TO FB_LABEL_2_0_0.INIT;
        FB_LABEL_2_0.INITO TO OUT_ANY_4.INIT;
        OUT_ANY_4.INITO TO FB_LABEL_2_1.INIT;
        FB_LABEL_2_1.INITO TO OUT_ANY_5.INIT;
        FB_LABEL_2_0_0.INITO TO OUT_ANY_6.INIT;
        OUT_ANY_6.INITO TO FB_LABEL_2_1_0.INIT;
        FB_LABEL_2_1_0.INITO TO OUT_ANY_7.INIT;
        OUT_ANY_5.INITO TO SUBSCRIBE_1_1.INIT;
        SUBSCRIBE_1_1.INITO TO SUBSCRIBE_1_2.INIT;
        OUT_ANY_7.INITO TO SUBSCRIBE_1_3.INIT;
        SUBSCRIBE_1_3.INITO TO SUBSCRIBE_1_4.INIT;
        SUBSCRIBE_1_1.IND TO STRING2STRING_3.REQ;
        STRING2STRING_3.CNF TO OUT_ANY_4.REQ;
        SUBSCRIBE_1_2.IND TO STRING2STRING_4.REQ;
        STRING2STRING_4.CNF TO OUT_ANY_5.REQ;
        SUBSCRIBE_1_3.IND TO STRING2STRING_5.REQ;
        STRING2STRING_5.CNF TO OUT_ANY_6.REQ;
        SUBSCRIBE_1_4.IND TO STRING2STRING_6.REQ;
        STRING2STRING_6.CNF TO OUT_ANY_7.REQ;
        START.COLD TO FB_LABEL_2.INIT;
        START.WARM TO FB_LABEL_2.INIT;
        START.COLD TO FB_LABEL_2_2.INIT;
        START.WARM TO FB_LABEL_2_2.INIT;
      END_CONNECTIONS
      DATA_CONNECTIONS
        SUBSCRIBE_1_1.RD_1 TO STRING2STRING_3.IN;
        STRING2STRING_3.OUT TO OUT_ANY_4.IN;
        SUBSCRIBE_1_2.RD_1 TO STRING2STRING_4.IN;
        STRING2STRING_4.OUT TO OUT_ANY_5.IN;
        SUBSCRIBE_1_3.RD_1 TO STRING2STRING_5.IN;
        STRING2STRING_5.OUT TO OUT_ANY_6.IN;
        SUBSCRIBE_1_4.RD_1 TO STRING2STRING_6.IN;
        STRING2STRING_6.OUT TO OUT_ANY_7.IN;
      END_CONNECTIONS
    END_RESOURCE
  END_DEVICE
  DEVICE RaspberryPI_1 : RaspberryPI(MGR_ID := "192.168.1.101:61499")
    {SET_ATTRIBUTE(Profile, HOLOBLOC)}
    RESOURCE EMB_RES : EMB_RES
      FBS
        UR2 : UR2(QI := 1);
        URMSGjudge : URMSGjudge(QI := 1);
        URMSGmonitoringRESULT : URMSGmonitoring(IVAL := ...);
        URClient : client(ID := UR, CONNECTTIME := T#3000ms, CHECKTIME := T#10ms);
        E_TimeOut_1 : E_TimeOut;
        E_TimeOut_3 : E_TimeOut;
        Camera : Camera(QI := 1);
        CameraMonitoringCMD : CameraMonitoring(IVAL := ...);
        CameraClient : client(ID := camera, CONNECTTIME := T#3000ms, CHECKTIME := T#10ms);
        E_TimeOut_4 : E_TimeOut;
        E_TimeOut_5 : E_TimeOut;
        SUBSCRIBE_2_0 : SUBSCRIBE_2(QI := 1, ID := %NetGateServerAddress%);
        SUBSCRIBE_0_0 : SUBSCRIBE_0(QI := 1, ID := %LifterPub%);
        SUBSCRIBE_0_1 : SUBSCRIBE_0(QI := 1, ID := %StopperPub%);
        PUBLISH_1 : PUBLISH_1(QI := 1, ID := %URPub1%);
        PUBLISH_0_1 : PUBLISH_0(QI := 1, ID := %URPub2%);
        SUBSCRIBE_2_1 : SUBSCRIBE_2(QI := 1, ID := %FindNextPub%);
        PUBLISH_1_3 : PUBLISH_1(QI := 1, ID := %URclient%);
        PUBLISH_1_4 : PUBLISH_1(QI := 1, ID := %Cameraclient%);
        CameraMonitoringRESULT : CameraMonitoring(IVAL := ...);
        URMSGmonitoringCMD : URMSGmonitoring(IVAL := ...);
        PUBLISH_1_5 : PUBLISH_1(QI := 1, ID := %URMoniteringCMD%);
        PUBLISH_1_6 : PUBLISH_1(QI := 1, ID := %URMoniteringRESULT%);
        PUBLISH_1_7 : PUBLISH_1(QI := 1, ID := %CameraMornitoringCMD%);
        PUBLISH_1_8 : PUBLISH_1(QI := 1, ID := %CameraMornitoringResult%);
      END_FBS
      EVENT_CONNECTIONS
        URMSGjudge.INITO TO UR2.INIT;
        URMSGjudge.URinPalletPosition TO UR2.URinPalletPosition;
        URMSGjudge.URinMaterialPosition TO UR2.URinMaterialPosition;
        URMSGjudge.GraspDone TO UR2.GraspDone;
        UR2.UROperation TO URClient.SEND;
        URClient.RECEIVED TO URMSGjudge.REQ;
        UR2.INITO TO Camera.INIT;
        UR2.TakePhoto TO Camera.TakePhoto;
        Camera.SendPhotoMSG TO UR2.RecvCameraMSG;
        URClient.INITO TO CameraClient.INIT;
        Camera.DoTakePhoto TO CameraClient.SEND;
        CameraClient.INITO TO URMSGjudge.INIT;
        CameraClient.RECEIVED TO Camera.RECVPhotoMSG;
        SUBSCRIBE_2_0.IND TO URClient.INIT;
        SUBSCRIBE_0_0.IND TO UR2.PalletIn;
        SUBSCRIBE_0_0.INITO TO SUBSCRIBE_0_1.INIT;
        SUBSCRIBE_0_1.IND TO UR2.INIT;
        SUBSCRIBE_0_1.INITO TO PUBLISH_1.INIT;
        UR2.SendPalletMSG TO PUBLISH_1.REQ;
        PUBLISH_1.INITO TO PUBLISH_0_1.INIT;
        UR2.UpdatePallet TO PUBLISH_0_1.REQ;
        PUBLISH_0_1.INITO TO SUBSCRIBE_2_1.INIT;
        SUBSCRIBE_2_1.IND TO UR2.URGrasp;
        SUBSCRIBE_2_1.INITO TO PUBLISH_1_3.INIT;
        URClient.STATE TO PUBLISH_1_3.REQ;
        PUBLISH_1_3.INITO TO PUBLISH_1_4.INIT;
        CameraClient.STATE TO PUBLISH_1_4.REQ;
        PUBLISH_1_4.INITO TO SUBSCRIBE_2_0.INIT;
        UR2.UROperation TO URMSGmonitoringRESULT.RESET;
        URClient.RECEIVED TO URMSGmonitoringRESULT.REQ;
        Camera.DoTakePhoto TO CameraMonitoringCMD.REQ;
        CameraClient.RECEIVED TO CameraMonitoringCMD.RESET;
        CameraClient.RECEIVED TO CameraMonitoringRESULT.REQ;
        Camera.DoTakePhoto TO CameraMonitoringRESULT.RESET;
        UR2.UROperation TO URMSGmonitoringCMD.REQ;
        URClient.RECEIVED TO URMSGmonitoringCMD.RESET;
        SUBSCRIBE_2_0.INITO TO PUBLISH_1_5.INIT;
        URMSGmonitoringCMD.CNF TO PUBLISH_1_5.REQ;
        PUBLISH_1_5.INITO TO PUBLISH_1_6.INIT;
        URMSGmonitoringRESULT.CNF TO PUBLISH_1_6.REQ;
        PUBLISH_1_6.INITO TO PUBLISH_1_7.INIT;
        CameraMonitoringCMD.CNF TO PUBLISH_1_7.REQ;
        PUBLISH_1_7.INITO TO PUBLISH_1_8.INIT;
        CameraMonitoringRESULT.CNF TO PUBLISH_1_8.REQ;
        START.COLD TO SUBSCRIBE_0_0.INIT;
        START.WARM TO SUBSCRIBE_0_0.INIT;
        UR2.INITO TO URMSGmonitoringCMD.RESET;
        UR2.INITO TO URMSGmonitoringRESULT.RESET;
        UR2.INITO TO CameraMonitoringCMD.RESET;
        UR2.INITO TO CameraMonitoringRESULT.RESET;
      END_CONNECTIONS
      DATA_CONNECTIONS
        UR2.toURMSG TO URClient.QI;
        URClient.QO TO URMSGjudge.URMSG;
        URClient.CheckTimeOut TO E_TimeOut_1.TimeOutSocket;
        URClient.ConnectTimeOut TO E_TimeOut_3.TimeOutSocket;
        UR2.TakePhotoNum TO Camera.PhotoNumIn;
        Camera.PhotoMSGOut1 TO UR2.PalletMSGIN;
        Camera.PhotoMSGOut2 TO UR2.MaterialMSG;
        Camera.PhotoNumOut TO CameraClient.QI;
        CameraClient.QO TO Camera.PhotoMSGIn;
        CameraClient.ConnectTimeOut TO E_TimeOut_4.TimeOutSocket;
        CameraClient.CheckTimeOut TO E_TimeOut_5.TimeOutSocket;
        SUBSCRIBE_2_0.RD_1 TO URClient.IP;
        SUBSCRIBE_2_0.RD_1 TO CameraClient.IP;
        SUBSCRIBE_2_0.RD_2 TO URClient.PORT;
        SUBSCRIBE_2_0.RD_2 TO CameraClient.PORT;
        UR2.PalletMSGOUT TO PUBLISH_1.SD_1;
        SUBSCRIBE_2_1.RD_1 TO UR2.URGraspModelPosition;
        SUBSCRIBE_2_1.RD_2 TO UR2.URGraspModelColour;
        URClient.RESULT TO PUBLISH_1_3.SD_1;
        CameraClient.RESULT TO PUBLISH_1_4.SD_1;
        URClient.QO TO URMSGmonitoringRESULT.MSGIN;
        Camera.PhotoNumOut TO CameraMonitoringCMD.MSGIN;
        CameraClient.QO TO CameraMonitoringRESULT.MSGIN;
        UR2.toURMSG TO URMSGmonitoringCMD.MSGIN;
        URMSGmonitoringCMD.MSGOUT TO PUBLISH_1_5.SD_1;
        URMSGmonitoringRESULT.MSGOUT TO PUBLISH_1_6.SD_1;
        CameraMonitoringCMD.MSGOUT TO PUBLISH_1_7.SD_1;
        CameraMonitoringRESULT.MSGOUT TO PUBLISH_1_8.SD_1;
      END_CONNECTIONS
    END_RESOURCE
  END_DEVICE
  DEVICE RaspberryPI_2 : RaspberryPI(MGR_ID := "192.168.1.102:61499")
    {SET_ATTRIBUTE(Profile, HOLOBLOC)}
    RESOURCE EMB_RES : EMB_RES
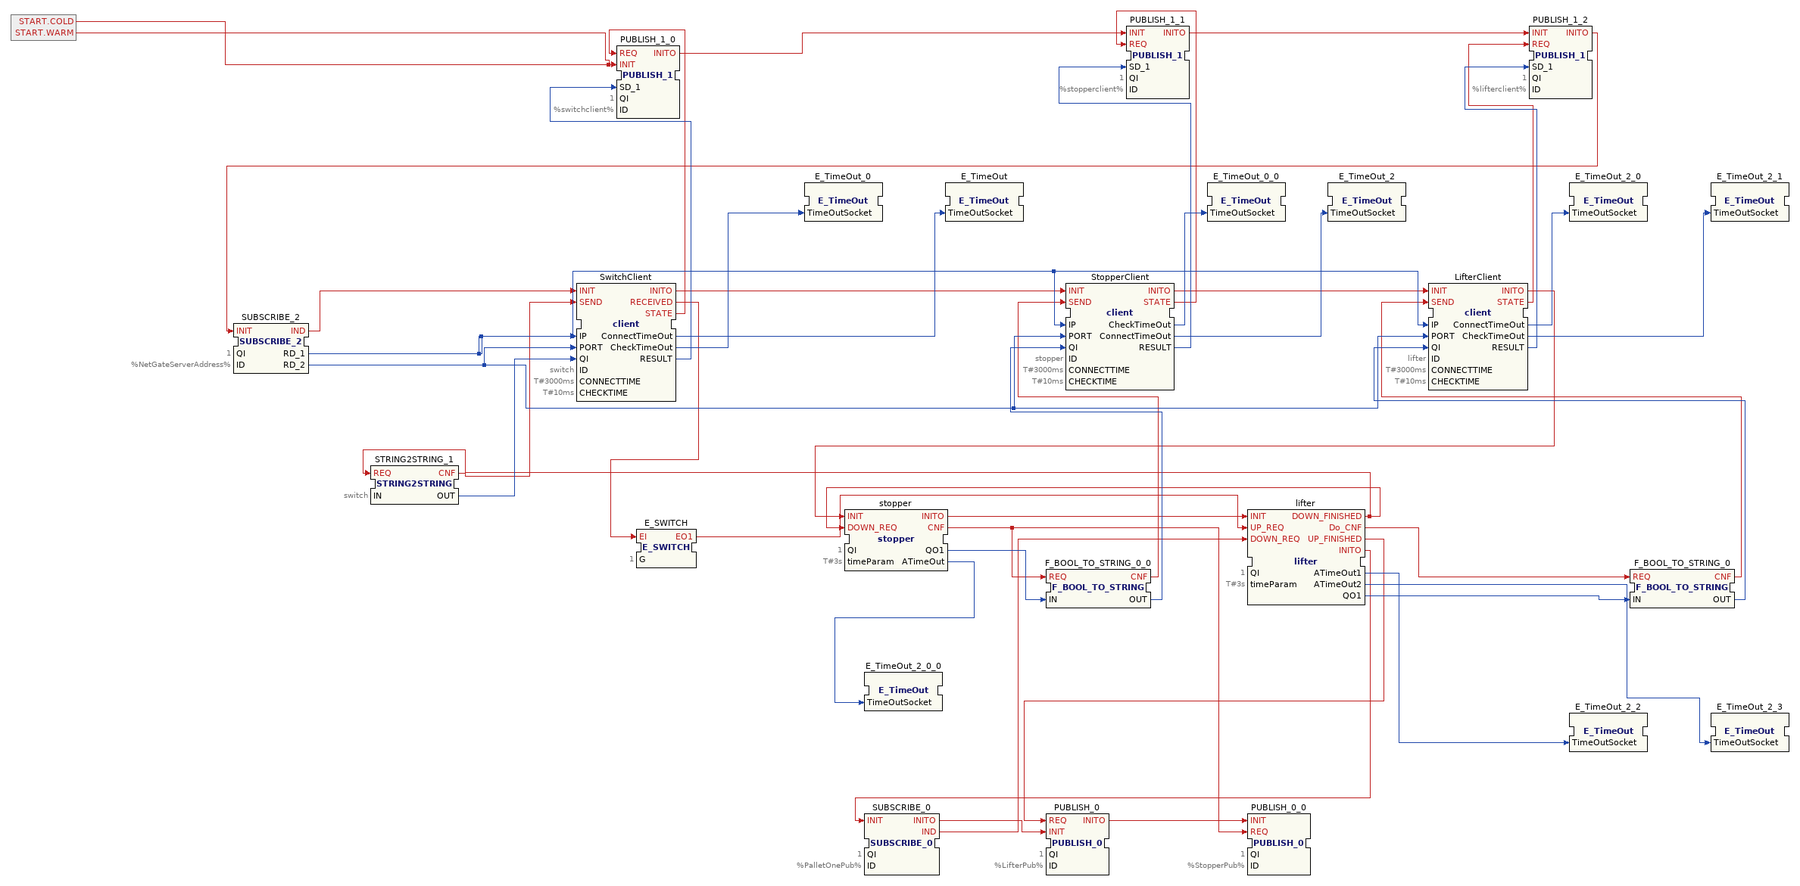
      FBS
        SwitchClient : client(ID := switch, CONNECTTIME := T#3000ms, CHECKTIME := T#10ms);
        E_TimeOut : E_TimeOut;
        E_TimeOut_0 : E_TimeOut;
        SUBSCRIBE_2 : SUBSCRIBE_2(QI := 1, ID := %NetGateServerAddress%);
        LifterClient : client(ID := lifter, CONNECTTIME := T#3000ms, CHECKTIME := T#10ms);
        E_TimeOut_0_0 : E_TimeOut;
        StopperClient : client(ID := stopper, CONNECTTIME := T#3000ms, CHECKTIME := T#10ms);
        E_TimeOut_2 : E_TimeOut;
        E_SWITCH : E_SWITCH(G := 1);
        stopper : stopper(QI := 1, timeParam := T#3s);
        lifter : lifter(QI := 1, timeParam := T#3s);
        E_TimeOut_2_0 : E_TimeOut;
        E_TimeOut_2_1 : E_TimeOut;
        E_TimeOut_2_2 : E_TimeOut;
        E_TimeOut_2_3 : E_TimeOut;
        F_BOOL_TO_STRING_0 : F_BOOL_TO_STRING;
        F_BOOL_TO_STRING_0_0 : F_BOOL_TO_STRING;
        E_TimeOut_2_0_0 : E_TimeOut;
        STRING2STRING_1 : STRING2STRING(IN := switch);
        PUBLISH_0 : PUBLISH_0(QI := 1, ID := %LifterPub%);
        SUBSCRIBE_0 : SUBSCRIBE_0(QI := 1, ID := %PalletOnePub%);
        PUBLISH_0_0 : PUBLISH_0(QI := 1, ID := %StopperPub%);
        PUBLISH_1_0 : PUBLISH_1(QI := 1, ID := %switchclient%);
        PUBLISH_1_1 : PUBLISH_1(QI := 1, ID := %stopperclient%);
        PUBLISH_1_2 : PUBLISH_1(QI := 1, ID := %lifterclient%);
      END_FBS
      EVENT_CONNECTIONS
        SUBSCRIBE_2.IND TO SwitchClient.INIT;
        SwitchClient.INITO TO StopperClient.INIT;
        StopperClient.INITO TO LifterClient.INIT;
        SwitchClient.RECEIVED TO E_SWITCH.EI;
        LifterClient.INITO TO stopper.INIT;
        stopper.INITO TO lifter.INIT;
        E_SWITCH.EO1 TO lifter.UP_REQ;
        lifter.DOWN_FINISHED TO stopper.DOWN_REQ;
        lifter.Do_CNF TO F_BOOL_TO_STRING_0.REQ;
        F_BOOL_TO_STRING_0.CNF TO LifterClient.SEND;
        stopper.CNF TO F_BOOL_TO_STRING_0_0.REQ;
        F_BOOL_TO_STRING_0_0.CNF TO StopperClient.SEND;
        lifter.DOWN_FINISHED TO STRING2STRING_1.REQ;
        STRING2STRING_1.CNF TO SwitchClient.SEND;
        lifter.UP_FINISHED TO PUBLISH_0.REQ;
        lifter.INITO TO SUBSCRIBE_0.INIT;
        SUBSCRIBE_0.INITO TO PUBLISH_0.INIT;
        SUBSCRIBE_0.IND TO lifter.DOWN_REQ;
        PUBLISH_0.INITO TO PUBLISH_0_0.INIT;
        stopper.CNF TO PUBLISH_0_0.REQ;
        SwitchClient.STATE TO PUBLISH_1_0.REQ;
        PUBLISH_1_0.INITO TO PUBLISH_1_1.INIT;
        StopperClient.STATE TO PUBLISH_1_1.REQ;
        PUBLISH_1_1.INITO TO PUBLISH_1_2.INIT;
        LifterClient.STATE TO PUBLISH_1_2.REQ;
        PUBLISH_1_2.INITO TO SUBSCRIBE_2.INIT;
        START.COLD TO PUBLISH_1_0.INIT;
        START.WARM TO PUBLISH_1_0.INIT;
      END_CONNECTIONS
      DATA_CONNECTIONS
        SwitchClient.ConnectTimeOut TO E_TimeOut.TimeOutSocket;
        SwitchClient.CheckTimeOut TO E_TimeOut_0.TimeOutSocket;
        SUBSCRIBE_2.RD_1 TO SwitchClient.IP;
        SUBSCRIBE_2.RD_2 TO SwitchClient.PORT;
        SUBSCRIBE_2.RD_1 TO LifterClient.IP;
        SUBSCRIBE_2.RD_2 TO LifterClient.PORT;
        SUBSCRIBE_2.RD_1 TO StopperClient.IP;
        SUBSCRIBE_2.RD_2 TO StopperClient.PORT;
        StopperClient.CheckTimeOut TO E_TimeOut_0_0.TimeOutSocket;
        StopperClient.ConnectTimeOut TO E_TimeOut_2.TimeOutSocket;
        LifterClient.ConnectTimeOut TO E_TimeOut_2_0.TimeOutSocket;
        LifterClient.CheckTimeOut TO E_TimeOut_2_1.TimeOutSocket;
        lifter.ATimeOut1 TO E_TimeOut_2_2.TimeOutSocket;
        lifter.ATimeOut2 TO E_TimeOut_2_3.TimeOutSocket;
        lifter.QO1 TO F_BOOL_TO_STRING_0.IN;
        F_BOOL_TO_STRING_0.OUT TO LifterClient.QI;
        stopper.QO1 TO F_BOOL_TO_STRING_0_0.IN;
        F_BOOL_TO_STRING_0_0.OUT TO StopperClient.QI;
        stopper.ATimeOut TO E_TimeOut_2_0_0.TimeOutSocket;
        STRING2STRING_1.OUT TO SwitchClient.QI;
        SwitchClient.RESULT TO PUBLISH_1_0.SD_1;
        StopperClient.RESULT TO PUBLISH_1_1.SD_1;
        LifterClient.RESULT TO PUBLISH_1_2.SD_1;
      END_CONNECTIONS
    END_RESOURCE
  END_DEVICE
  MAPPINGS
    HMI.FB_LABEL ON FBRT_WINDOW.ConnectSet.FB_LABEL;
    HMI.FB_LABEL_0 ON FBRT_WINDOW.ConnectSet.FB_LABEL_0;
    HMI.IN_ANY ON FBRT_WINDOW.ConnectSet.IN_ANY;
    HMI.IN_ANY_0 ON FBRT_WINDOW.ConnectSet.IN_ANY_0;
    HMI.PUBLISH_2 ON FBRT_WINDOW.ConnectSet.PUBLISH_2;
    HMI.STRING2STRING ON FBRT_WINDOW.ConnectSet.STRING2STRING;
    HMI.STRING2STRING_0 ON FBRT_WINDOW.ConnectSet.STRING2STRING_0;
    HMI.IN_EVENT ON FBRT_WINDOW.ConnectSet.IN_EVENT;
    HMI.FB_LABEL_1 ON FBRT_WINDOW.ClientConnection.FB_LABEL_1;
    HMI.FB_LABEL_1_0 ON FBRT_WINDOW.ClientConnection.FB_LABEL_1_0;
    HMI.FB_LABEL_1_1 ON FBRT_WINDOW.ClientConnection.FB_LABEL_1_1;
    HMI.FB_LABEL_1_2 ON FBRT_WINDOW.ClientConnection.FB_LABEL_1_2;
    HMI.FB_LABEL_1_3 ON FBRT_WINDOW.ClientConnection.FB_LABEL_1_3;
    HMI.OUT_ANY ON FBRT_WINDOW.ClientConnection.OUT_ANY;
    HMI.OUT_ANY_0 ON FBRT_WINDOW.ClientConnection.OUT_ANY_0;
    HMI.OUT_ANY_1 ON FBRT_WINDOW.ClientConnection.OUT_ANY_1;
    HMI.OUT_ANY_2 ON FBRT_WINDOW.ClientConnection.OUT_ANY_2;
    HMI.OUT_ANY_3 ON FBRT_WINDOW.ClientConnection.OUT_ANY_3;
    HMI.SUBSCRIBE_1_0 ON FBRT_WINDOW.ClientConnection.SUBSCRIBE_1_0;
    HMI.SUBSCRIBE_1_0_0 ON FBRT_WINDOW.ClientConnection.SUBSCRIBE_1_0_0;
    HMI.SUBSCRIBE_1_0_1 ON FBRT_WINDOW.ClientConnection.SUBSCRIBE_1_0_1;
    HMI.SUBSCRIBE_1_0_2 ON FBRT_WINDOW.ClientConnection.SUBSCRIBE_1_0_2;
    HMI.SUBSCRIBE_1_0_3 ON FBRT_WINDOW.ClientConnection.SUBSCRIBE_1_0_3;
    HMI.STRING2STRING_2 ON FBRT_WINDOW.ClientConnection.STRING2STRING_2;
    HMI.STRING2STRING_2_0 ON FBRT_WINDOW.ClientConnection.STRING2STRING_2_0;
    HMI.STRING2STRING_2_1 ON FBRT_WINDOW.ClientConnection.STRING2STRING_2_1;
    HMI.STRING2STRING_2_2 ON FBRT_WINDOW.ClientConnection.STRING2STRING_2_2;
    HMI.STRING2STRING_2_3 ON FBRT_WINDOW.ClientConnection.STRING2STRING_2_3;
    HMI.FB_LABEL_2 ON FBRT_WINDOW.MachineState.FB_LABEL_2;
    HMI.FB_LABEL_2_0 ON FBRT_WINDOW.MachineState.FB_LABEL_2_0;
    HMI.FB_LABEL_2_1 ON FBRT_WINDOW.MachineState.FB_LABEL_2_1;
    HMI.FB_LABEL_2_2 ON FBRT_WINDOW.MachineState.FB_LABEL_2_2;
    HMI.FB_LABEL_2_0_0 ON FBRT_WINDOW.MachineState.FB_LABEL_2_0_0;
    HMI.FB_LABEL_2_1_0 ON FBRT_WINDOW.MachineState.FB_LABEL_2_1_0;
    HMI.OUT_ANY_4 ON FBRT_WINDOW.MachineState.OUT_ANY_4;
    HMI.OUT_ANY_5 ON FBRT_WINDOW.MachineState.OUT_ANY_5;
    HMI.OUT_ANY_6 ON FBRT_WINDOW.MachineState.OUT_ANY_6;
    HMI.OUT_ANY_7 ON FBRT_WINDOW.MachineState.OUT_ANY_7;
    HMI.SUBSCRIBE_1_1 ON FBRT_WINDOW.MachineState.SUBSCRIBE_1_1;
    HMI.SUBSCRIBE_1_2 ON FBRT_WINDOW.MachineState.SUBSCRIBE_1_2;
    HMI.SUBSCRIBE_1_3 ON FBRT_WINDOW.MachineState.SUBSCRIBE_1_3;
    HMI.SUBSCRIBE_1_4 ON FBRT_WINDOW.MachineState.SUBSCRIBE_1_4;
    HMI.STRING2STRING_3 ON FBRT_WINDOW.MachineState.STRING2STRING_3;
    HMI.STRING2STRING_4 ON FBRT_WINDOW.MachineState.STRING2STRING_4;
    HMI.STRING2STRING_5 ON FBRT_WINDOW.MachineState.STRING2STRING_5;
    HMI.STRING2STRING_6 ON FBRT_WINDOW.MachineState.STRING2STRING_6;
    SwitchStopperLifter.SwitchClient ON RaspberryPI_2.EMB_RES.SwitchClient;
    SwitchStopperLifter.E_TimeOut ON RaspberryPI_2.EMB_RES.E_TimeOut;
    SwitchStopperLifter.E_TimeOut_0 ON RaspberryPI_2.EMB_RES.E_TimeOut_0;
    SwitchStopperLifter.SUBSCRIBE_2 ON RaspberryPI_2.EMB_RES.SUBSCRIBE_2;
    SwitchStopperLifter.LifterClient ON RaspberryPI_2.EMB_RES.LifterClient;
    SwitchStopperLifter.E_TimeOut_0_0 ON RaspberryPI_2.EMB_RES.E_TimeOut_0_0;
    SwitchStopperLifter.StopperClient ON RaspberryPI_2.EMB_RES.StopperClient;
    SwitchStopperLifter.E_TimeOut_2 ON RaspberryPI_2.EMB_RES.E_TimeOut_2;
    SwitchStopperLifter.E_SWITCH ON RaspberryPI_2.EMB_RES.E_SWITCH;
    SwitchStopperLifter.stopper ON RaspberryPI_2.EMB_RES.stopper;
    SwitchStopperLifter.lifter ON RaspberryPI_2.EMB_RES.lifter;
    SwitchStopperLifter.E_TimeOut_2_0 ON RaspberryPI_2.EMB_RES.E_TimeOut_2_0;
    SwitchStopperLifter.E_TimeOut_2_1 ON RaspberryPI_2.EMB_RES.E_TimeOut_2_1;
    SwitchStopperLifter.E_TimeOut_2_2 ON RaspberryPI_2.EMB_RES.E_TimeOut_2_2;
    SwitchStopperLifter.E_TimeOut_2_3 ON RaspberryPI_2.EMB_RES.E_TimeOut_2_3;
    SwitchStopperLifter.F_BOOL_TO_STRING_0 ON RaspberryPI_2.EMB_RES.F_BOOL_TO_STRING_0;
    SwitchStopperLifter.F_BOOL_TO_STRING_0_0 ON RaspberryPI_2.EMB_RES.F_BOOL_TO_STRING_0_0;
    SwitchStopperLifter.E_TimeOut_2_0_0 ON RaspberryPI_2.EMB_RES.E_TimeOut_2_0_0;
    SwitchStopperLifter.STRING2STRING_1 ON RaspberryPI_2.EMB_RES.STRING2STRING_1;
    SwitchStopperLifter.PUBLISH_0 ON RaspberryPI_2.EMB_RES.PUBLISH_0;
    SwitchStopperLifter.SUBSCRIBE_0 ON RaspberryPI_2.EMB_RES.SUBSCRIBE_0;
    SwitchStopperLifter.PUBLISH_0_0 ON RaspberryPI_2.EMB_RES.PUBLISH_0_0;
    SwitchStopperLifter.PUBLISH_1_0 ON RaspberryPI_2.EMB_RES.PUBLISH_1_0;
    SwitchStopperLifter.PUBLISH_1_1 ON RaspberryPI_2.EMB_RES.PUBLISH_1_1;
    SwitchStopperLifter.PUBLISH_1_2 ON RaspberryPI_2.EMB_RES.PUBLISH_1_2;
    URCamera.UR2 ON RaspberryPI_1.EMB_RES.UR2;
    URCamera.URMSGjudge ON RaspberryPI_1.EMB_RES.URMSGjudge;
    URCamera.URMSGmonitoringRESULT ON RaspberryPI_1.EMB_RES.URMSGmonitoringRESULT;
    URCamera.URClient ON RaspberryPI_1.EMB_RES.URClient;
    URCamera.E_TimeOut_1 ON RaspberryPI_1.EMB_RES.E_TimeOut_1;
    URCamera.E_TimeOut_3 ON RaspberryPI_1.EMB_RES.E_TimeOut_3;
    URCamera.Camera ON RaspberryPI_1.EMB_RES.Camera;
    URCamera.CameraMonitoringCMD ON RaspberryPI_1.EMB_RES.CameraMonitoringCMD;
    URCamera.CameraClient ON RaspberryPI_1.EMB_RES.CameraClient;
    URCamera.E_TimeOut_4 ON RaspberryPI_1.EMB_RES.E_TimeOut_4;
    URCamera.E_TimeOut_5 ON RaspberryPI_1.EMB_RES.E_TimeOut_5;
    URCamera.SUBSCRIBE_2_0 ON RaspberryPI_1.EMB_RES.SUBSCRIBE_2_0;
    URCamera.SUBSCRIBE_0_0 ON RaspberryPI_1.EMB_RES.SUBSCRIBE_0_0;
    URCamera.SUBSCRIBE_0_1 ON RaspberryPI_1.EMB_RES.SUBSCRIBE_0_1;
    URCamera.PUBLISH_1 ON RaspberryPI_1.EMB_RES.PUBLISH_1;
    URCamera.PUBLISH_0_1 ON RaspberryPI_1.EMB_RES.PUBLISH_0_1;
    URCamera.SUBSCRIBE_2_1 ON RaspberryPI_1.EMB_RES.SUBSCRIBE_2_1;
    URCamera.PUBLISH_1_3 ON RaspberryPI_1.EMB_RES.PUBLISH_1_3;
    URCamera.PUBLISH_1_4 ON RaspberryPI_1.EMB_RES.PUBLISH_1_4;
    URCamera.URMSGmonitoringCMD ON RaspberryPI_1.EMB_RES.URMSGmonitoringCMD;
    URCamera.CameraMonitoringRESULT ON RaspberryPI_1.EMB_RES.CameraMonitoringRESULT;
    URCamera.PUBLISH_1_5 ON RaspberryPI_1.EMB_RES.PUBLISH_1_5;
    URCamera.PUBLISH_1_6 ON RaspberryPI_1.EMB_RES.PUBLISH_1_6;
    URCamera.PUBLISH_1_7 ON RaspberryPI_1.EMB_RES.PUBLISH_1_7;
    URCamera.PUBLISH_1_8 ON RaspberryPI_1.EMB_RES.PUBLISH_1_8;
    DataBaseOperation.sqlUpdateMaterial ON FORTE_PC.EMB_RES.sqlUpdateMaterial;
    DataBaseOperation.splitCameraInfo ON FORTE_PC.EMB_RES.splitCameraInfo;
    DataBaseOperation.findNext ON FORTE_PC.EMB_RES.findNext;
    DataBaseOperation.palletOne ON FORTE_PC.EMB_RES.palletOne;
    DataBaseOperation.SUBSCRIBE_0_2 ON FORTE_PC.EMB_RES.SUBSCRIBE_0_2;
    DataBaseOperation.SUBSCRIBE_1 ON FORTE_PC.EMB_RES.SUBSCRIBE_1;
    DataBaseOperation.PUBLISH_2_0 ON FORTE_PC.EMB_RES.PUBLISH_2_0;
    DataBaseOperation.PUBLISH_0_2 ON FORTE_PC.EMB_RES.PUBLISH_0_2;
  END_MAPPINGS
  SEGMENTS
    Ethernet : Ethernet;
  END_SEGMENTS
  LINKS
    RaspberryPI_1 => Ethernet;
    RaspberryPI_2 => Ethernet;
    FORTE_PC => Ethernet;
    FBRT_WINDOW => Ethernet;
  END_LINKS
END_SYSTEM
